Staubli VAL3: getObjectOffset.pgx

program getObjectOffset(num x_nConvNum (dimensions=1), num x_nIdx (dimensions=1), num& x_nObjectOffset[] (dimensions=1), num& x_nError[] (dimensions=1))
  local point l_pDummy
  local point l_pPoint
begin
  switch x_nConvNum
    case 0
      call cnv0:getObjectOffset(x_nIdx,x_nObjectOffset,x_nError)
    break
    case 1
      call cnv1:getObjectOffset(x_nIdx,x_nObjectOffset,x_nError)
    break
  endSwitch
end
